(*			
	EVERDE sp. z o.o.
	Rafał Osajda		22.01.2025		TC 4026.13		wer. 0.0.0.1
	Sterowanie lampką
*)
FUNCTION_BLOCK FB_Lamp EXTENDS FB_BaseComponent IMPLEMENTS ITF_Lamp
VAR
	bOut							AT %Q*	: BOOL;		// Lampka
END_VAR

(*			
	EVERDE sp. z o.o.
	Rafał Osajda		05.02.2025		TC 4026.13		wer. 0.0.0.1
	Sterowanie swieceniem lampki - włącz/wyłącz
*)
METHOD Control
VAR_INPUT
	bIN	: BOOL;
END_VAR
IF (bIN) THEN
	THIS^.SetOn ();
ELSE
	THIS^.SetOff ();
END_IF
END_METHOD

(*			
	EVERDE sp. z o.o.
	Rafał Osajda		05.02.2025		TC 4026.13		wer. 0.0.0.1
	Zwraca czy lampka wlaczona
*)
METHOD IsActive : BOOL
IsActive					:= THIS^.bOut;
END_METHOD

(*			
	EVERDE sp. z o.o.
	Rafał Osajda		05.02.2025		TC 4026.13		wer. 0.0.0.1
	Wylacza lampke
*)
METHOD SetOff
THIS^.bOut				:= FALSE;
END_METHOD

(*			
	EVERDE sp. z o.o.
	Rafał Osajda		05.02.2025		TC 4026.13		wer. 0.0.0.1
	Wlacza lampke
*)
METHOD SetOn
THIS^.bOut				:= TRUE;
END_METHOD

END_FUNCTION_BLOCK

(* stored: Version 1.1.0.1
   POU FB_Lamp: Id {30c1ff06-6578-49b3-9061-1ee463c72ccc}, SpecialFunc None
   Method Control: Id {844f4e13-0894-473a-87fc-66d05adf3dd4}
   Method IsActive: Id {d932e6d0-a12f-4bd1-9eb7-c6f588f2fc10}
   Method SetOff: Id {a3ef5c87-3683-438c-8b1e-bffac6b99dbd}
   Method SetOn: Id {5d58c598-4dc3-4264-8e5b-5d3cc338857a} *)
